TYPE ST_FanucCNCEventDetails :
STRUCT
	AxesMask : ST_FanucCNCEventAxesMask;
	Category : BYTE;
	No : UINT;
END_STRUCT
END_TYPE

(* stored: Version 1.1.0.1, ProductVersion 3.1.4024.12
   DUT ST_FanucCNCEventDetails: Id {24b7c173-ec86-41c3-a846-fe2335fe8c18} *)
